Omron CX-Programmer project NewProject (CX-Programmer 9.61)

# PLC LAMPU_GANTIAN: CP1L M

## Global symbols (name address type ; comment)
0.00 BOOL  ; PB START
0.01 BOOL  ; PB STOP
100.00 BOOL  ; SELF HOLDING
100.01 BOOL  ; LAMPU1
100.02 BOOL  ; LAMPU2
100.03 BOOL  ; LAMPU3
100.04 BOOL  ; LAMPU4
100.05 BOOL  ; LAMPU5
100.06 BOOL  ; LAMPU6
100.07 BOOL  ; LAMPU7
100.08 BOOL  ; LAMPU8
T0000 BOOL  ; TIMER1
T0000 BOOL  ; TIMER1

## Program NewProgram1 (cyclic task 0)

### Section Section1

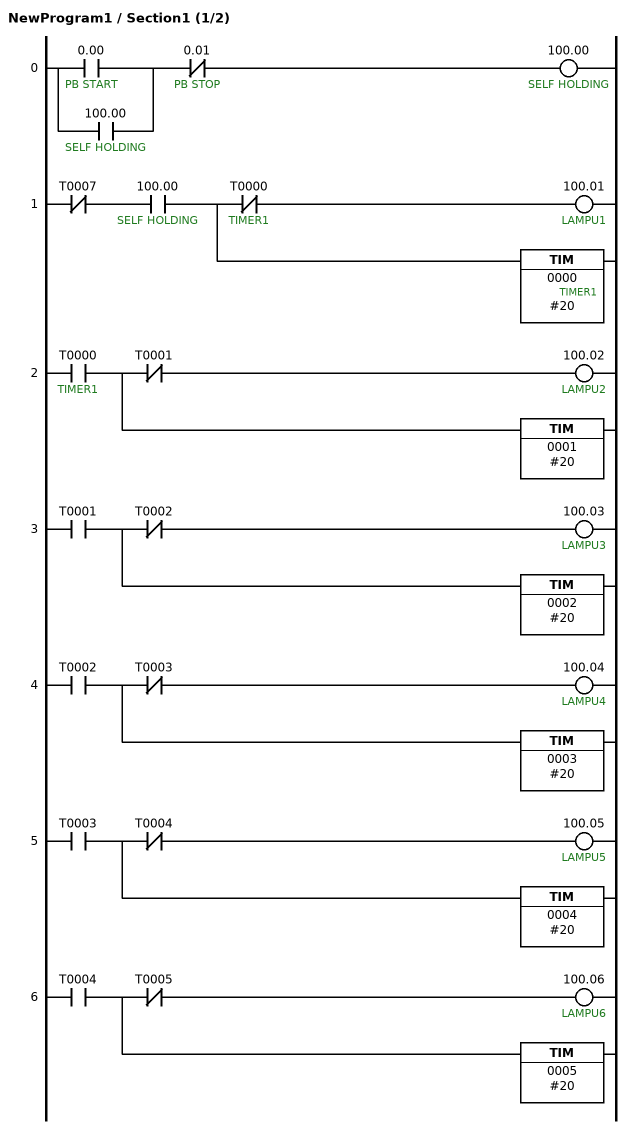
; rung 0
LD 0.00  ; PB START
OR 100.00  ; SELF HOLDING
ANDNOT 0.01  ; PB STOP
OUT 100.00  ; SELF HOLDING
; rung 1
LDNOT T0007
AND 100.00  ; SELF HOLDING
OUT TR0
ANDNOT T0000  ; TIMER1
OUT 100.01  ; LAMPU1
LD TR0
TIM 0000 #20  ; TIMER1
; rung 2
LD T0000  ; TIMER1
OUT TR0
ANDNOT T0001
OUT 100.02  ; LAMPU2
LD TR0
TIM 0001 #20
; rung 3
LD T0001
OUT TR0
ANDNOT T0002
OUT 100.03  ; LAMPU3
LD TR0
TIM 0002 #20
; rung 4
LD T0002
OUT TR0
ANDNOT T0003
OUT 100.04  ; LAMPU4
LD TR0
TIM 0003 #20
; rung 5
LD T0003
OUT TR0
ANDNOT T0004
OUT 100.05  ; LAMPU5
LD TR0
TIM 0004 #20
; rung 6
LD T0004
OUT TR0
ANDNOT T0005
OUT 100.06  ; LAMPU6
LD TR0
TIM 0005 #20

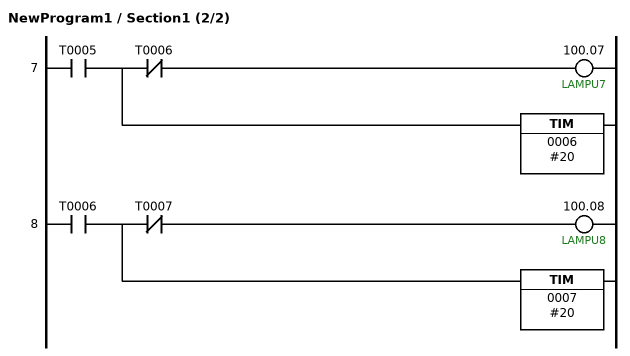
; rung 7
LD T0005
OUT TR0
ANDNOT T0006
OUT 100.07  ; LAMPU7
LD TR0
TIM 0006 #20
; rung 8
LD T0006
OUT TR0
ANDNOT T0007
OUT 100.08  ; LAMPU8
LD TR0
TIM 0007 #20

### Section END
; rung 0
END(001)